TYPE WcStateInputToggleBase_F68C23A9 :
STRUCT
END_STRUCT
END_TYPE

(* stored: Version 1.1.0.1, ProductVersion 3.1.4024.9
   DUT WcStateInputToggleBase_F68C23A9: Id {7c859641-68fc-02f1-2c7c-625b912a7315} *)
